// TwinCAT 3 PLC project TcControl
// Title: TcControl
// Company: Roald
// Author: Roald Ruiter
// ProjectVersion: 0.5.2
// Description: PID control function blocks
// ProgramVersion: 3.1.4023.0
// libraries:
//   Tc2_Standard, * (Beckhoff Automation GmbH)
//   Tc2_System, * (Beckhoff Automation GmbH)
//   Tc3_Module, * (Beckhoff Automation GmbH)
//   TcUnit, * (www.tcunit.org)
// project tree:
//   / Derivative.TcPOU, IBaseSignal.TcIO, IController.TcIO, IDifferentiable.TcIO, InstancePath.TcPOU, InfiniteImpulseResponse.TcPOU, IOut.TcIO, ISignal.TcIO, Millisecond.TcDUT, Signal.TcPOU, PidController.TcPOU, PidParameters.TcDUT, PlcTask.TcTTO, RemoveProjectName.TcPOU
//   Tests/ Derivative_Tests.TcPOU, InfiniteImpulseResponse_Tests.TcPOU, Signal_Tests.TcPOU, Pid_Tests.TcPOU, UnitTests.TcPOU
// real-time tasks:
//   TASK PlcTask: cycle T#10ms, priority 21, ADS port 351

CONFIGURATION TcControl
    RESOURCE PLC ON TwinCAT3
        TASK PlcTask(INTERVAL := T#10ms, PRIORITY := 21);
        PROGRAM UnitTests WITH PlcTask : UnitTests;
    END_RESOURCE
END_CONFIGURATION

// ---- Millisecond.TcDUT
TYPE Millisecond : LREAL; END_TYPE

// ---- PidParameters.TcDUT
TYPE PidParameters :
STRUCT
    Kp : LREAL;
    Ki : LREAL;
    Kd : LREAL;
END_STRUCT
END_TYPE

// ---- IBaseSignal.TcIO
INTERFACE IBaseSignal EXTENDS IOut

METHOD Control : IOut
VAR_INPUT
    setpoint : LREAL;
END_VAR
END_METHOD

METHOD Update : ISignal
VAR_INPUT
    value : LREAL;
END_VAR
END_METHOD

END_INTERFACE

// ---- IController.TcIO
INTERFACE IController EXTENDS IOut

METHOD Update : IOut
VAR_INPUT
    setpoint : LREAL;
    actual : LREAL;
END_VAR
END_METHOD

END_INTERFACE

// ---- IDifferentiable.TcIO
INTERFACE IDifferentiable EXTENDS IOut

METHOD Control: IOut
VAR_INPUT
    setpoint : LREAL;
END_VAR
END_METHOD

METHOD Iir : IBaseSignal
VAR_INPUT
    decay : LREAL;
END_VAR
END_METHOD

METHOD Update : ISignal
VAR_INPUT
    value : LREAL;
END_VAR
END_METHOD

END_INTERFACE

// ---- IOut.TcIO
INTERFACE IOut

PROPERTY Out : LREAL
GET
END_GET
END_PROPERTY

END_INTERFACE

// ---- ISignal.TcIO
INTERFACE ISignal EXTENDS IOut

METHOD Control : IOut
VAR_INPUT
    setpoint : LREAL;
END_VAR
END_METHOD

METHOD Differentiate : IDifferentiable
VAR_INPUT
    deltaTime : Millisecond;
END_VAR
END_METHOD

METHOD Iir : IBaseSignal
VAR_INPUT
    decay : LREAL;
END_VAR
END_METHOD

METHOD Update : ISignal
VAR_INPUT
    value : LREAL;
END_VAR
END_METHOD

END_INTERFACE

// ---- Tests/UnitTests.TcPOU
PROGRAM UnitTests
VAR
    pidTests : Pid_Tests;
    infiniteImpluseResponseTests : InfiniteImpulseResponse_Tests;
    derivativeTests : Derivative_Tests;
    signalTests : Signal_Tests;
END_VAR

TcUnit.RUN();

END_PROGRAM

// ---- Tests/Pid_Tests.TcPOU
FUNCTION_BLOCK Pid_Tests EXTENDS FB_TestSuite
VAR
    delta : LREAL := 1E-5;
END_VAR

OnlyProportionalPart();
OnlyPropotionalPartRunTwiceWithDifferentInputs();
OnlyIntegralPart();
OnlyIntegralPartSetPreviousIntegralPartBefore();
OnlyDifferentialPart();
OnlyDifferentialPartWithDiffLimit();
DifferentCycleTimesSameOutputIntegralPart();
DifferentCycleTimesSameOutputDifferentialPart();
DivideByZeroCycleTimeCheck();

METHOD DifferentCycleTimesSameOutputDifferentialPart
VAR_INST
    Pfast : PidController;
    Pslow : PidController;
    parameters : PidParameters := (Kd:=1);
    i : INT;
END_VAR
TEST('DifferentCycleTimesSameOutputDifferentialPart');

Pfast(parameters:=parameters, cycleTime:=1);
FOR i := 1 TO 4 DO
    Pfast.Update(setpoint:=3, actual:=2 + i * 0.25);
END_FOR

Pslow(parameters:=parameters, cycleTime:=2);
FOR i := 1 TO 2 DO
    Pslow.Update(setpoint:=3, actual:=2 + i * 0.5);
END_FOR

AssertEquals_LREAL(
    Expected:=Pslow.Out,
    Actual:=Pfast.Out,
    Delta:=delta,
    Message:='Slow and fast pid should give the same result'
);

TcUnit.TEST_FINISHED();
END_METHOD

METHOD DifferentCycleTimesSameOutputIntegralPart
VAR_INST
    Pfast : PidController;
    Pslow : PidController;
    parameters : PidParameters := (Ki:=1);
END_VAR
TEST('DifferentCycleTimesSameOutputIntegralPart');

Pfast(parameters:=parameters, cycleTime:=1);
Pfast.Update(setpoint:=3, actual:=2);
Pfast.Update(setpoint:=3, actual:=2);
Pslow(parameters:=parameters, cycleTime:=2);
Pslow.Update(setpoint:=3, actual:=2);

AssertEquals_LREAL(
    Expected:=Pslow.Out,
    Actual:=Pfast.Out,
    Delta:=delta,
    Message:='Slow and fast pid should give the same result'
);

TcUnit.TEST_FINISHED();
END_METHOD

METHOD DivideByZeroCycleTimeCheck
VAR_INST
    P : PidController;
END_VAR
TcUnit.TEST('DivideByZeroCycleTimeCheck');

P(cycleTime:=0);
P.Update(setpoint:=1, actual:=1);

//Should not cause an exception

TcUnit.TEST_FINISHED();
END_METHOD

METHOD OnlyDifferentialPart
VAR_INST
    P : PidController;
    parameters : PidParameters := (Kd:=0.01);
END_VAR
TcUnit.TEST('OnlyDifferentialPart');

P(parameters:=parameters);
P.Update(setpoint:=10, actual:=6);
AssertEquals_LREAL(
    Expected:=0.04,
    Actual:=P.Out,
    Delta:=delta,
    Message:='Pid output run 1 not correct'
);

P.Update(setpoint:=10, actual:=8);
AssertEquals_LREAL(
    Expected:=-0.02,
    Actual:=P.Out,
    Delta:=delta,
    Message:='Pid output run 2 not correct'
);

TcUnit.TEST_FINISHED();
END_METHOD

METHOD OnlyDifferentialPartWithDiffLimit
VAR_INST
    P : PidController;
    parameters : PidParameters := (Kd:=0.01);
END_VAR
TcUnit.TEST('OnlyDifferentialPartWithDiffLimit');

P.DifferentialPartLimit := 3;
P(parameters:=parameters);
P.Update(setpoint:=10, actual:=6);
AssertEquals_LREAL(
    Expected:=0,
    Actual:=P.Out,
    Delta:=delta,
    Message:='Pid output run 1 not correct'
);

P.Update(setpoint:=10, actual:=8);
AssertEquals_LREAL(
    Expected:=-0.02,
    Actual:=P.Out,
    Delta:=delta,
    Message:='Pid output run 2 not correct'
);

TcUnit.TEST_FINISHED();
END_METHOD

METHOD OnlyIntegralPart
VAR_INST
    P : PidController := (cycleTime:=1);
    parameters : PidParameters := (Ki:=0.25);
END_VAR
TcUnit.TEST('OnlyIntegralPart');

P(parameters:=parameters);
P.Update(setpoint:=10, actual:=6);
AssertEquals_LREAL(
    Expected:=1,
    Actual:=P.Out,
    Delta:=delta,
    Message:='Pid output run 1 not correct'
);

P.Update(setpoint:=10, actual:=8);
AssertEquals_LREAL(
    Expected:=1.5,
    Actual:=P.Out,
    Delta:=delta,
    Message:='Pid output run 2 not correct'
);

TcUnit.TEST_FINISHED();
END_METHOD

METHOD OnlyIntegralPartSetPreviousIntegralPartBefore
VAR_INST
    P : PidController := (cycleTime:=1);
    parameters : PidParameters := (Ki:=0.25);
END_VAR
TcUnit.TEST('OnlyIntegralPartSetPreviousIntegralPartBefore');

P.PreviousIntegralPart := 3;
P(parameters:=parameters);
P.Update(setpoint:=10, actual:=6);
AssertEquals_LREAL(
    Expected:=4,
    Actual:=P.Out,
    Delta:=delta,
    Message:='Pid output run 1 not correct'
);

P.Update(setpoint:=10, actual:=8);
AssertEquals_LREAL(
    Expected:=4.5,
    Actual:=P.Out,
    Delta:=delta,
    Message:='Pid output run 2 not correct'
);

TcUnit.TEST_FINISHED();
END_METHOD

METHOD OnlyProportionalPart
VAR_INST
    P : PidController;
    parameters : PidParameters := (Kp:=5);
END_VAR
TcUnit.TEST('OnlyProportionalPart');

P(parameters:=parameters);
P.Update(setpoint:=10, actual:=5);

AssertEquals_LREAL(Expected:=25, Actual:=P.Out, Delta:=delta, Message:='Pid output not correct');

TcUnit.TEST_FINISHED();
END_METHOD

METHOD OnlyPropotionalPartRunTwiceWithDifferentInputs
VAR_INST
    P : PidController;
    parameters : PidParameters := (Kp:=2);
END_VAR
TcUnit.TEST('OnlyPropotionalPartRunTwiceWithDifferentInputs');

P(parameters:=parameters);
P.Update(setpoint:=3, actual:=4.5);

AssertEquals_LREAL(
    Expected:=-3,
    Actual:=P.Out,
    Delta:=delta,
    Message:='Pid output after run 1 not correct'
);

P.Update(setpoint:=-8, actual:=-6);

AssertEquals_LREAL(
    Expected:=-4,
    Actual:=P.Out,
    Delta:=delta,
    Message:='Pid output after run 2 not correct'
);

TcUnit.TEST_FINISHED();
END_METHOD

END_FUNCTION_BLOCK

// ---- PidController.TcPOU
FUNCTION_BLOCK PidController EXTENDS InstancePath IMPLEMENTS IController, IOut
VAR_INPUT
    parameters : PidParameters;
    cycleTime : Millisecond := 1;
END_VAR
VAR
    _error : LREAL;
    _previousError : LREAL;
    _deltaError : LREAL;
    _proportionalPart : LREAL;
    _integralPart : LREAL;
    _previousIntegralPart : LREAL;
    _differentialPart : LREAL;
    _differentialPartLimit : LREAL;
    _out : LREAL;
END_VAR

(* Limit the differential part. Convenient when the output is calculated for the first time.
The limit prevents it from having a very large value after the first call.*)
PROPERTY DifferentialPartLimit : LREAL
SET
_differentialPartLimit := DifferentialPartLimit;
END_SET
END_PROPERTY

PROPERTY Out : LREAL
GET
Out := _out;
END_GET
END_PROPERTY

(* Set previous integral part on first call. Prevents integrator term for needing to build up. *)
PROPERTY PreviousIntegralPart : LREAL
SET
_previousIntegralPart := PreviousIntegralPart;
END_SET
END_PROPERTY

METHOD Update : IOut
VAR_INPUT
    setpoint : LREAL;
    actual : LREAL;
END_VAR
_error := setpoint - actual;

_proportionalPart := parameters.Kp * _error;

_integralPart := _previousIntegralPart + parameters.Ki * _error * cycleTime;
_previousIntegralPart := _integralPart;

IF cycleTime <> 0 THEN
    _deltaError := (_error - _previousError) / cycleTime;
ELSE
    ADSLOGSTR(
        msgCtrlMask:=ADSLOG_MSGTYPE_ERROR,
        msgFmtStr:='%s: Enter a cycletime > 0!',
        strArg:=_path
    );
END_IF
IF _differentialPartLimit = 0 OR _deltaError <= _differentialPartLimit THEN
    _differentialPart := _deltaError * parameters.Kd;
END_IF
_previousError := _error;

_out := _proportionalPart + _integralPart + _differentialPart;
END_METHOD

END_FUNCTION_BLOCK

// ---- InstancePath.TcPOU
(* Get the instance path of a function block
Source: https://kassymdorsel.com/blog/2021-01-06-automatic-instance-path-for-error-log-identification
*)
{attribute 'reflection'}
FUNCTION_BLOCK InstancePath
VAR
    {attribute 'instance-path'}
    {attribute 'noinit'}
    _path : Tc2_System.T_MaxString;
END_VAR

METHOD FB_init : BOOL
VAR_INPUT
    bInitRetains : BOOL; // if TRUE, the retain variables are initialized (warm start / cold start)
    bInCopyCode : BOOL; // if TRUE, the instance afterwards gets moved into the copy code (online change)
END_VAR
_path := RemoveProjectName(_path);
END_METHOD

END_FUNCTION_BLOCK

// ---- RemoveProjectName.TcPOU
(* Removes project name from string
Source: https://kassymdorsel.com/blog/2021-01-06-automatic-instance-path-for-error-log-identification
*)
FUNCTION RemoveProjectName : T_MaxString
VAR_INPUT
    path : T_MaxString;
END_VAR

RemoveProjectName := DELETE(
    path,
    LEN(TwinCAT_SystemInfoVarList._AppInfo.ProjectName) +
        FIND(path, TwinCAT_SystemInfoVarList._AppInfo.ProjectName),
    1
);

END_FUNCTION

// ---- Tests/InfiniteImpulseResponse_Tests.TcPOU
FUNCTION_BLOCK InfiniteImpulseResponse_Tests EXTENDS FB_TestSuite
VAR
    delta : LREAL := 1e-5;
END_VAR

CalculateImpulseResponse();
CalculateStepResponse();

METHOD CalculateImpulseResponse
VAR_INST
    iir : InfiniteImpulseResponse;
    i : DINT;
    decay : LREAL := 0.9;
    step : LREAL := 1;
END_VAR
TcUnit.TEST('CalculateImpulseResponse');

iir(new:=step, decay:=decay);
FOR i := 0 TO 9 DO
    AssertEquals_LREAL(
        Expected:=(1 - decay) * EXPT(decay, i),
        Actual:=iir.Out,
        Message:=CONCAT('Fail at i=', TO_STRING(i)),
        Delta:=delta
    );
    iir(new:=0);
END_FOR

TcUnit.TEST_FINISHED();
END_METHOD

METHOD CalculateStepResponse
VAR_INST
    iir : InfiniteImpulseResponse;
    i : DINT;
    decay : LREAL := 0.95;
    step : LREAL := 5;
    expected : ARRAY[0..9] OF LREAL := [0.25,
        0.4875,
        0.71313,
        0.92747,
        1.1311,
        1.32454,
        1.50831,
        1.6829,
        1.84875,
        2.00632];
END_VAR
TcUnit.TEST('CalculateStepResponse');

FOR i := 0 TO 9 DO
    iir(new:=step, decay:=decay);
    AssertEquals_LREAL(
        Expected:=expected[i],
        Actual:=iir.Out,
        Message:=CONCAT('Fail at i=', TO_STRING(i)),
        Delta:=delta
    );
END_FOR

TcUnit.TEST_FINISHED();
END_METHOD

END_FUNCTION_BLOCK

// ---- InfiniteImpulseResponse.TcPOU
(* Low pass Infinite Impulse Response (IIR) filter*)
FUNCTION_BLOCK InfiniteImpulseResponse IMPLEMENTS IOut
VAR_INPUT
    new : LREAL;
    decay : LREAL;
END_VAR
VAR
    _previous : LREAL;
    _out : LREAL;
END_VAR

_out := _previous * decay + new * (1 - decay);
_previous := _out;

PROPERTY Out : LREAL
GET
Out := _out;
END_GET
END_PROPERTY

END_FUNCTION_BLOCK

// ---- Tests/Derivative_Tests.TcPOU
FUNCTION_BLOCK Derivative_Tests EXTENDS FB_TestSuite
VAR
    delta : LREAL := 1e-5;
END_VAR

FirstCallDerivateiveIsZero();
CalculatederivateOnSecondCall();
PreventZeroDivisionException();

METHOD CalculatederivateOnSecondCall
VAR_INST
    d : Derivative;
END_VAR
TEST('CalculatederivateOnSecondCall');

d(value:=1, deltatime:=1);
d(value:=2, deltatime:=1);

AssertEquals_LREAL(Expected:=1, Actual:=d.Out, Delta:=delta, Message:='derivative not correct');

TcUnit.TEST_FINISHED();
END_METHOD

METHOD FirstCallDerivateiveIsZero
VAR_INST
    d : Derivative;
END_VAR
TEST('FirstCallDerivateiveIsZero');

d(value:=1, deltatime:=1);

AssertEquals_LREAL(Expected:=0, Actual:=d.Out, Delta:=delta, Message:='derivative not correct');

TcUnit.TEST_FINISHED();
END_METHOD

METHOD PreventZeroDivisionException
VAR_INST
    d : Derivative;
    path : STRING;
END_VAR
TEST('PreventZeroDivisionException');

d(deltatime:=0);
d(deltatime:=0);

// should not crash plc
path := d._path;

TcUnit.TEST_FINISHED();
END_METHOD

END_FUNCTION_BLOCK

// ---- Derivative.TcPOU
{attribute 'reflection'}
FUNCTION_BLOCK Derivative EXTENDS InstancePath IMPLEMENTS IOut
VAR_INPUT
    value : LREAL;
    deltaTime : Millisecond;
END_VAR
VAR
    _out : LREAL;
    _previousValue : LREAL;
    _firstCall : BOOL := TRUE;
END_VAR

IF _firstCall THEN
    _firstCall := FALSE;
ELSE
    IF deltaTime <> 0 THEN
        _out := (value - _previousValue) / deltaTime;
    ELSE
        ADSLOGSTR(
            msgCtrlMask:=ADSLOG_MSGTYPE_ERROR,
            msgFmtStr:='%s: Enter a delta time > 0!',
            strArg:=_path
        );
    END_IF
END_IF
_previousValue := value;

PROPERTY Out : LREAL
GET
Out := _out;
END_GET
END_PROPERTY

END_FUNCTION_BLOCK

// ---- Tests/Signal_Tests.TcPOU
FUNCTION_BLOCK Signal_Tests EXTENDS FB_TestSuite
VAR_INPUT
    delta : LREAL := 1E-5;
    si : Signal;
END_VAR

OnlyMeasurementShouldReturnSameValue();
TakeDerivativeOfMeasurement();
ApplyIirFilterOnSignal();
ApplyDiffAndIirOnSignal();
TestPidController();

METHOD ApplyDiffAndIirOnSignal
VAR_INST
    signal : Signal;
END_VAR
TEST('ApplyDiffAndIirOnSignal');

signal.Update(value:=7).Differentiate(deltaTime:=1).Iir(decay:=0.5);
AssertEquals_LREAL(
    Expected:=0,
    Actual:=signal.Out,
    Delta:=delta,
    Message:='Output step 1 not correct'
);

signal.Update(value:=8).Differentiate(deltaTime:=1).Iir(decay:=0.5);
AssertEquals_LREAL(
    Expected:=0.5,
    Actual:=signal.Out,
    Delta:=delta,
    Message:='Output step 2 not correct'
);

signal.Update(value:=9).Differentiate(deltaTime:=1).Iir(decay:=0.5);
AssertEquals_LREAL(
    Expected:=0.75,
    Actual:=signal.Out,
    Delta:=delta,
    Message:='Output step 3 not correct'
);

TcUnit.TEST_FINISHED();
END_METHOD

METHOD ApplyIirFilterOnSignal
VAR_INST
    signal : Signal;
    actual : LREAL;
END_VAR
TEST('ApplyIirFilterOnSignal');

signal.Update(value:=1.4).Iir(decay:=0.5);
AssertEquals_LREAL(Expected:=0.7, Actual:=signal.Out, Delta:=delta, Message:='Output not correct');

actual := signal.Update(value:=8.6).Iir(decay:=0.5).Out;
AssertEquals_LREAL(Expected:=4.65, Actual:=actual, Delta:=delta, Message:='Output not correct');

TcUnit.TEST_FINISHED();
END_METHOD

METHOD OnlyMeasurementShouldReturnSameValue : LREAL
VAR_INST
    signal : Signal;
END_VAR
TEST('OnlyMeasurementShouldReturnSameValue');

signal.Update(value:=1.23);

AssertEquals_LREAL(
    Expected:=1.23,
    Actual:=signal.Out,
    Delta:=delta,
    Message:='Output not correct'
);

TcUnit.TEST_FINISHED();
END_METHOD

METHOD TakeDerivativeOfMeasurement : LREAL
VAR_INST
    signal : Signal;
    actual : LREAL;
END_VAR
TEST('TakeDerivativeOfMeasurement');

actual := signal.Update(value:=1).Differentiate(deltaTime:=1).Out;
AssertEquals_LREAL(
    Expected:=0,
    Actual:=actual,
    Delta:=delta,
    Message:='Derivative after first step not correct'
);

actual := signal.Update(value:=2).Differentiate(deltaTime:=1).Out;
AssertEquals_LREAL(
    Expected:=1,
    Actual:=actual,
    Delta:=delta,
    Message:='Derivative after second step not correct'
);

TcUnit.TEST_FINISHED();
END_METHOD

METHOD TestPidController
VAR_INST
    _signal : Signal;
    parameters : PidParameters := (Kp:=2, Ki:=0.25, Kd:=0.5);
    pid : PidController;
END_VAR
TEST('TestPidController');

pid(parameters:=parameters, cycleTime:=1);
_signal.Controller := pid;
_signal.Update(3).Control(setpoint:=4);

AssertEquals_LREAL(
    Expected:=2.75,
    Actual:=_signal.Out,
    Delta:=delta,
    Message:='Pid output not correct after cycle 1'
);

_signal.Update(3.5).Control(setpoint:=4);

AssertEquals_LREAL(
    Expected:=1.125,
    Actual:=_signal.Out,
    Delta:=delta,
    Message:='Pid output not correct after cycle 2'
);

TcUnit.TEST_FINISHED();
END_METHOD

END_FUNCTION_BLOCK

// ---- Signal.TcPOU
FUNCTION_BLOCK Signal EXTENDS InstancePath IMPLEMENTS IBaseSignal, IDifferentiable, ISignal
VAR
    _out : LREAL;
    _derivative : Derivative;
    _iir : InfiniteImpulseResponse;
    _controller : IController;
END_VAR

METHOD Control : IOut
VAR_INPUT
    setpoint : LREAL;
END_VAR
IF _controller <> 0 THEN
    _controller.Update(setpoint:=setpoint, actual:=THIS^.Out);
    _out := _controller.Out;
    Control := THIS^;
ELSE
    ADSLOGSTR(
        msgCtrlMask:=ADSLOG_MSGTYPE_ERROR,
        msgFmtStr:='%s: Assign a controller before calling this method.',
        strArg:=_path
    );
END_IF
END_METHOD

PROPERTY Controller : IController
SET
_controller := Controller;
END_SET
END_PROPERTY

METHOD Differentiate : IDifferentiable
VAR_INPUT
    deltaTime : Millisecond;
END_VAR
_derivative(value:=THIS^.Out, deltaTime:=deltaTime);
_out := _derivative.Out;
Differentiate := THIS^;
END_METHOD

METHOD Iir : IBaseSignal
VAR_INPUT
    decay : LREAL;
END_VAR
_iir(new:=THIS^.Out, decay:=decay);
_out := _iir.Out;
Iir := THIS^;
END_METHOD

PROPERTY Out : LREAL
GET
OUT := _out;
END_GET
END_PROPERTY

METHOD Update : ISignal
VAR_INPUT
    value : LREAL;
END_VAR
_out := value;
Update := THIS^;
END_METHOD

END_FUNCTION_BLOCK
